Staubli VAL3: deleteItem.pgx

public program deleteItem(num x_nIndex)
begin
end
